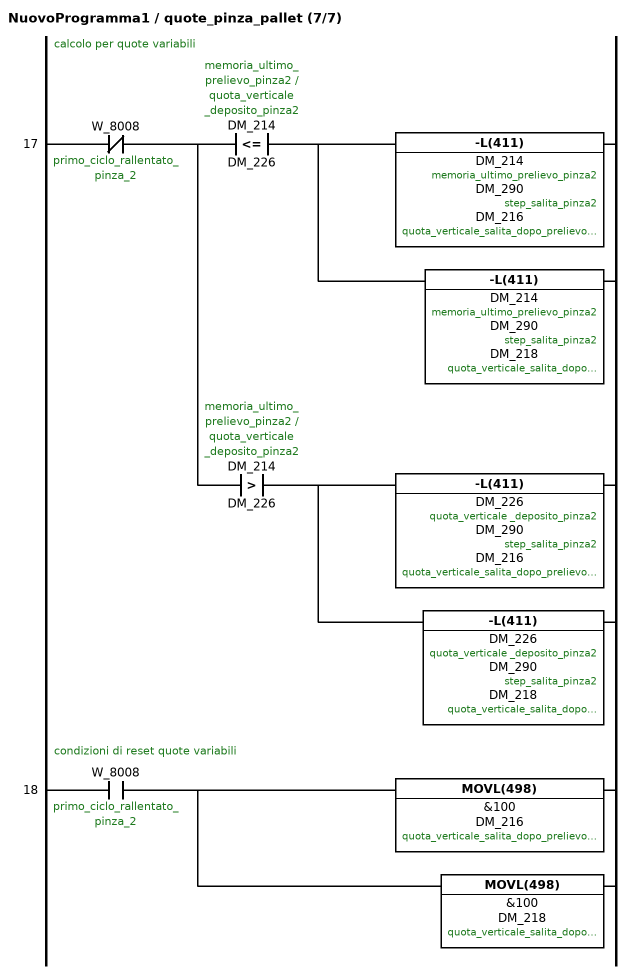
; [picture p96: NuovoProgramma1 / quote_pinza_pallet, rungs 17-18]
; rung 17: calcolo per quote variabili
LDNOT W_8008  ; primo_ciclo_rallentato_pinza_2
OUT TR0
AND<=SL(318) DM_214 DM_226  ; memoria_ultimo_prelievo_pinza2, quota_verticale _deposito_pinza2
-L(411) DM_214 DM_290 DM_216  ; memoria_ultimo_prelievo_pinza2, step_salita_pinza2, quota_verticale_salita_dopo_prelievo_pinza2
-L(411) DM_214 DM_290 DM_218  ; memoria_ultimo_prelievo_pinza2, step_salita_pinza2, quota_verticale_salita_dopo_deposito_pinza2
LD TR0
AND>SL(323) DM_214 DM_226  ; memoria_ultimo_prelievo_pinza2, quota_verticale _deposito_pinza2
-L(411) DM_226 DM_290 DM_216  ; quota_verticale _deposito_pinza2, step_salita_pinza2, quota_verticale_salita_dopo_prelievo_pinza2
-L(411) DM_226 DM_290 DM_218  ; quota_verticale _deposito_pinza2, step_salita_pinza2, quota_verticale_salita_dopo_deposito_pinza2
; rung 18: condizioni di reset quote variabili
LD W_8008  ; primo_ciclo_rallentato_pinza_2
MOVL(498) &100 DM_216  ; quota_verticale_salita_dopo_prelievo_pinza2
MOVL(498) &100 DM_218  ; quota_verticale_salita_dopo_deposito_pinza2

### Section cambi_pallet

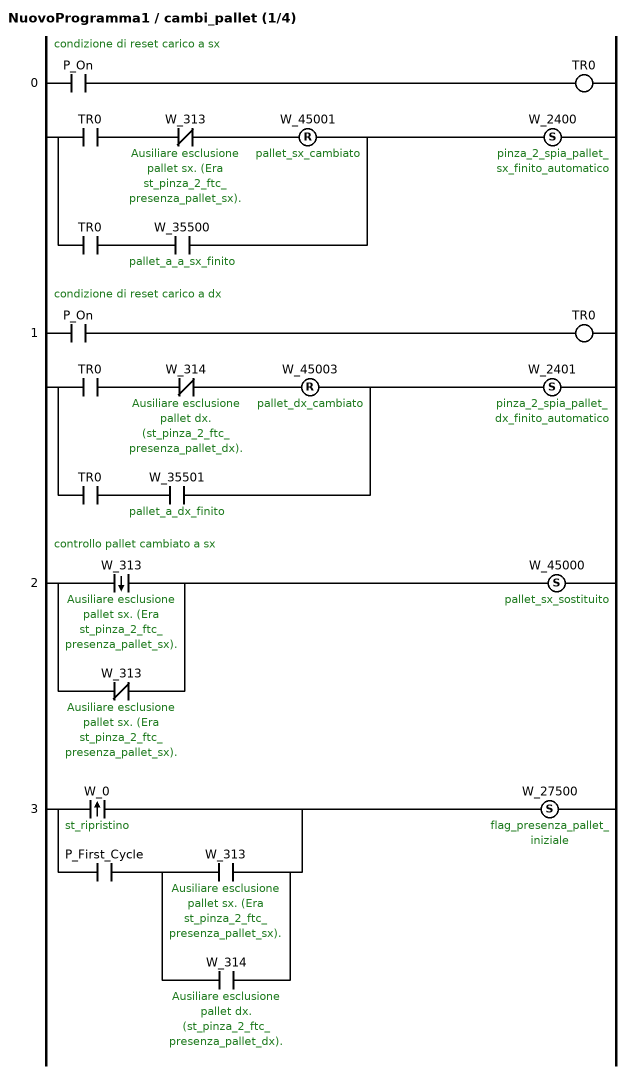
; rung 0: condizione di reset carico a sx
LD P_On
OUT TR0
ANDNOT W_313  ; Ausiliare esclusione pallet sx. (Era st_pinza_2_ftc_presenza_pallet_sx).
RSET W_45001  ; pallet_sx_cambiato
LD TR0
AND W_35500  ; pallet_a_a_sx_finito
ORLD
SET W_2400  ; pinza_2_spia_pallet_sx_finito_automatico
; rung 1: condizione di reset carico a dx
LD P_On
OUT TR0
ANDNOT W_314  ; Ausiliare esclusione pallet dx. (st_pinza_2_ftc_presenza_pallet_dx).
RSET W_45003  ; pallet_dx_cambiato
LD TR0
AND W_35501  ; pallet_a_dx_finito
ORLD
SET W_2401  ; pinza_2_spia_pallet_dx_finito_automatico
; rung 2: controllo pallet cambiato a sx
%LD W_313  ; Ausiliare esclusione pallet sx. (Era st_pinza_2_ftc_presenza_pallet_sx).
ORNOT W_313  ; Ausiliare esclusione pallet sx. (Era st_pinza_2_ftc_presenza_pallet_sx).
SET W_45000  ; pallet_sx_sostituito
; rung 3
@LD W_0  ; st_ripristino
LD P_First_Cycle
LD W_313  ; Ausiliare esclusione pallet sx. (Era st_pinza_2_ftc_presenza_pallet_sx).
OR W_314  ; Ausiliare esclusione pallet dx. (st_pinza_2_ftc_presenza_pallet_dx).
ANDLD
ORLD
SET W_27500  ; flag_presenza_pallet_iniziale

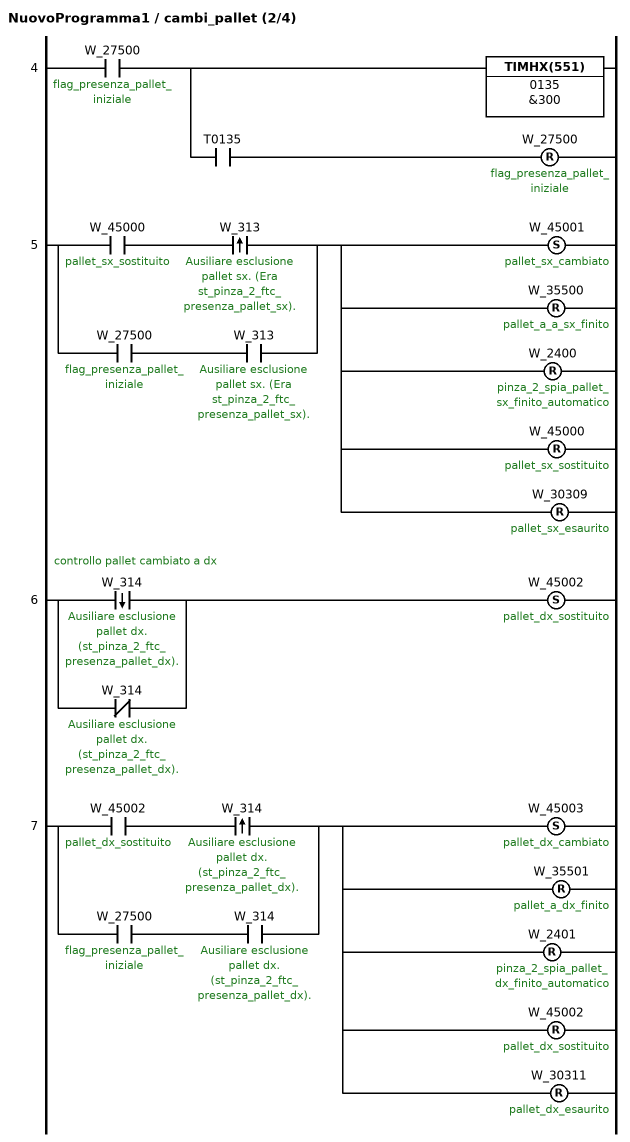
; rung 4
LD W_27500  ; flag_presenza_pallet_iniziale
TIMHX(551) 0135 &300
AND T0135
RSET W_27500  ; flag_presenza_pallet_iniziale
; rung 5
LD W_45000  ; pallet_sx_sostituito
@AND W_313  ; Ausiliare esclusione pallet sx. (Era st_pinza_2_ftc_presenza_pallet_sx).
LD W_27500  ; flag_presenza_pallet_iniziale
AND W_313  ; Ausiliare esclusione pallet sx. (Era st_pinza_2_ftc_presenza_pallet_sx).
ORLD
SET W_45001  ; pallet_sx_cambiato
RSET W_35500  ; pallet_a_a_sx_finito
RSET W_2400  ; pinza_2_spia_pallet_sx_finito_automatico
RSET W_45000  ; pallet_sx_sostituito
RSET W_30309  ; pallet_sx_esaurito
; rung 6: controllo pallet cambiato a dx
%LD W_314  ; Ausiliare esclusione pallet dx. (st_pinza_2_ftc_presenza_pallet_dx).
ORNOT W_314  ; Ausiliare esclusione pallet dx. (st_pinza_2_ftc_presenza_pallet_dx).
SET W_45002  ; pallet_dx_sostituito
; rung 7
LD W_45002  ; pallet_dx_sostituito
@AND W_314  ; Ausiliare esclusione pallet dx. (st_pinza_2_ftc_presenza_pallet_dx).
LD W_27500  ; flag_presenza_pallet_iniziale
AND W_314  ; Ausiliare esclusione pallet dx. (st_pinza_2_ftc_presenza_pallet_dx).
ORLD
SET W_45003  ; pallet_dx_cambiato
RSET W_35501  ; pallet_a_dx_finito
RSET W_2401  ; pinza_2_spia_pallet_dx_finito_automatico
RSET W_45002  ; pallet_dx_sostituito
RSET W_30311  ; pallet_dx_esaurito

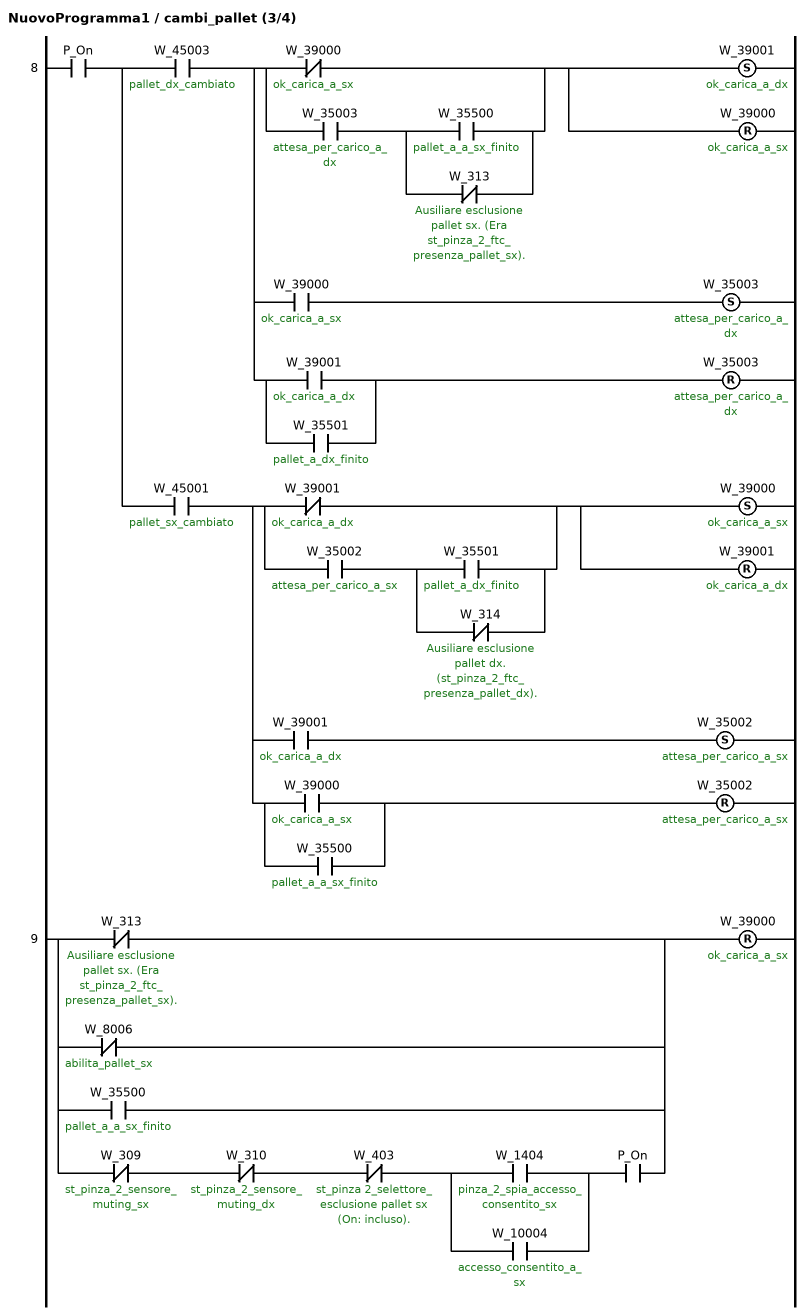
; rung 8
LD P_On
OUT TR0
AND W_45003  ; pallet_dx_cambiato
OUT TR1
LDNOT W_39000  ; ok_carica_a_sx
LD W_35003  ; attesa_per_carico_a_dx
LD W_35500  ; pallet_a_a_sx_finito
ORNOT W_313  ; Ausiliare esclusione pallet sx. (Era st_pinza_2_ftc_presenza_pallet_sx).
ANDLD
ORLD
ANDLD
SET W_39001  ; ok_carica_a_dx
RSET W_39000  ; ok_carica_a_sx
LD TR1
AND W_39000  ; ok_carica_a_sx
SET W_35003  ; attesa_per_carico_a_dx
LD TR1
LD W_39001  ; ok_carica_a_dx
OR W_35501  ; pallet_a_dx_finito
ANDLD
RSET W_35003  ; attesa_per_carico_a_dx
LD TR0
AND W_45001  ; pallet_sx_cambiato
OUT TR0
LDNOT W_39001  ; ok_carica_a_dx
LD W_35002  ; attesa_per_carico_a_sx
LD W_35501  ; pallet_a_dx_finito
ORNOT W_314  ; Ausiliare esclusione pallet dx. (st_pinza_2_ftc_presenza_pallet_dx).
ANDLD
ORLD
ANDLD
SET W_39000  ; ok_carica_a_sx
RSET W_39001  ; ok_carica_a_dx
LD TR0
AND W_39001  ; ok_carica_a_dx
SET W_35002  ; attesa_per_carico_a_sx
LD TR0
LD W_39000  ; ok_carica_a_sx
OR W_35500  ; pallet_a_a_sx_finito
ANDLD
RSET W_35002  ; attesa_per_carico_a_sx
; rung 9
LDNOT W_313  ; Ausiliare esclusione pallet sx. (Era st_pinza_2_ftc_presenza_pallet_sx).
ORNOT W_8006  ; abilita_pallet_sx
OR W_35500  ; pallet_a_a_sx_finito
LDNOT W_309  ; st_pinza_2_sensore_muting_sx
ANDNOT W_310  ; st_pinza_2_sensore_muting_dx
ANDNOT W_403  ; st_pinza 2_selettore_esclusione pallet sx (On: incluso).
LD W_1404  ; pinza_2_spia_accesso_consentito_sx
OR W_10004  ; accesso_consentito_a_sx
ANDLD
AND P_On
ORLD
RSET W_39000  ; ok_carica_a_sx

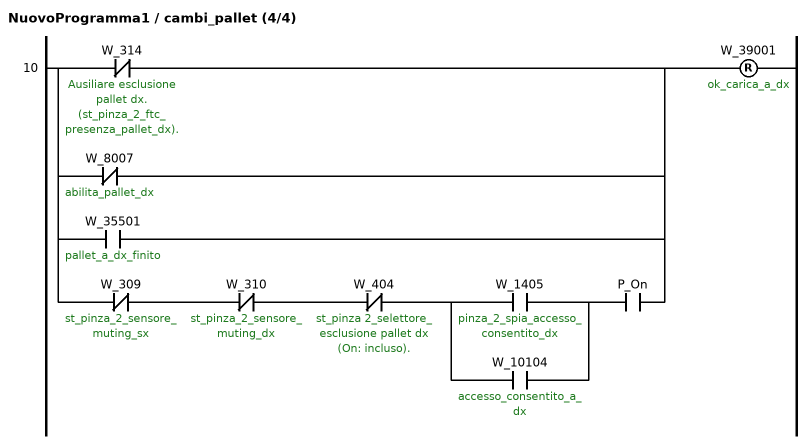
; rung 10
LDNOT W_314  ; Ausiliare esclusione pallet dx. (st_pinza_2_ftc_presenza_pallet_dx).
ORNOT W_8007  ; abilita_pallet_dx
OR W_35501  ; pallet_a_dx_finito
LDNOT W_309  ; st_pinza_2_sensore_muting_sx
ANDNOT W_310  ; st_pinza_2_sensore_muting_dx
ANDNOT W_404  ; st_pinza 2_selettore_esclusione pallet dx (On: incluso).
LD W_1405  ; pinza_2_spia_accesso_consentito_dx
OR W_10104  ; accesso_consentito_a_dx
ANDLD
AND P_On
ORLD
RSET W_39001  ; ok_carica_a_dx

### Section accessi

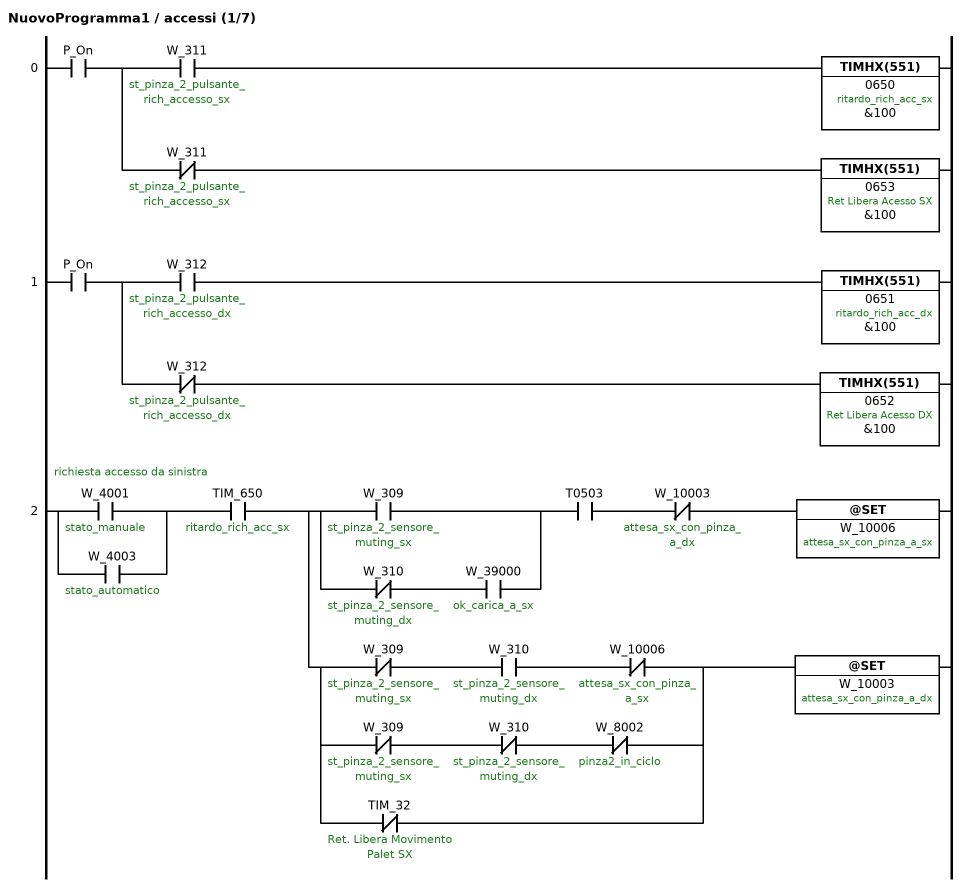
; rung 0
LD P_On
OUT TR0
AND W_311  ; st_pinza_2_pulsante_rich_accesso_sx
TIMHX(551) 0650 &100  ; ritardo_rich_acc_sx
LD TR0
ANDNOT W_311  ; st_pinza_2_pulsante_rich_accesso_sx
TIMHX(551) 0653 &100  ; Ret Libera Acesso SX
; rung 1
LD P_On
OUT TR0
AND W_312  ; st_pinza_2_pulsante_rich_accesso_dx
TIMHX(551) 0651 &100  ; ritardo_rich_acc_dx
LD TR0
ANDNOT W_312  ; st_pinza_2_pulsante_rich_accesso_dx
TIMHX(551) 0652 &100  ; Ret Libera Acesso DX
; rung 2: richiesta accesso da sinistra
LD W_4001  ; stato_manuale
OR W_4003  ; stato_automatico
AND TIM_650  ; ritardo_rich_acc_sx
OUT TR0
LD W_309  ; st_pinza_2_sensore_muting_sx
LDNOT W_310  ; st_pinza_2_sensore_muting_dx
AND W_39000  ; ok_carica_a_sx
ORLD
ANDLD
AND T0503
ANDNOT W_10003  ; attesa_sx_con_pinza_a_dx
@SET W_10006  ; attesa_sx_con_pinza_a_sx
LD TR0
LDNOT W_309  ; st_pinza_2_sensore_muting_sx
AND W_310  ; st_pinza_2_sensore_muting_dx
ANDNOT W_10006  ; attesa_sx_con_pinza_a_sx
LDNOT W_309  ; st_pinza_2_sensore_muting_sx
ANDNOT W_310  ; st_pinza_2_sensore_muting_dx
ANDNOT W_8002  ; pinza2_in_ciclo
ORLD
ORNOT TIM_32  ; Ret. Libera Movimento Palet SX
ANDLD
@SET W_10003  ; attesa_sx_con_pinza_a_dx

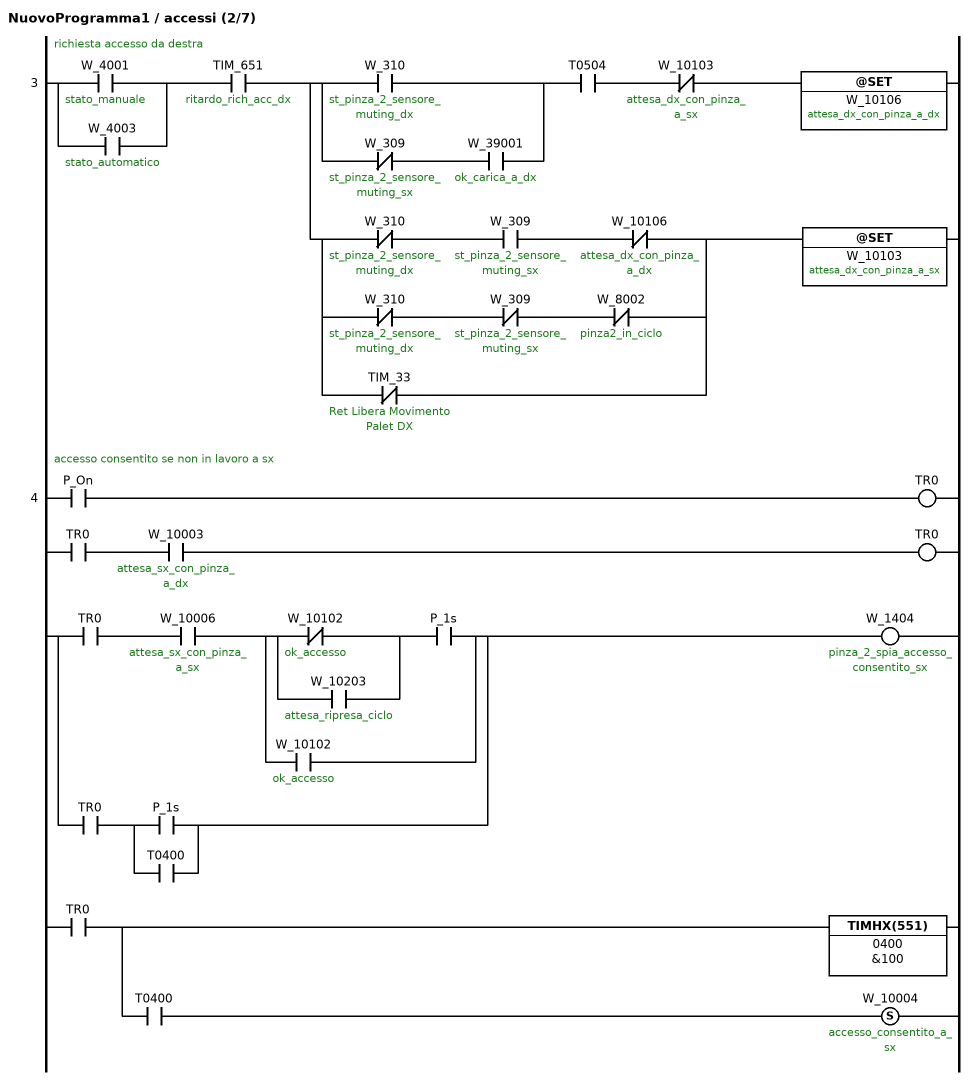
; rung 3: richiesta accesso da destra
LD W_4001  ; stato_manuale
OR W_4003  ; stato_automatico
AND TIM_651  ; ritardo_rich_acc_dx
OUT TR0
LD W_310  ; st_pinza_2_sensore_muting_dx
LDNOT W_309  ; st_pinza_2_sensore_muting_sx
AND W_39001  ; ok_carica_a_dx
ORLD
ANDLD
AND T0504
ANDNOT W_10103  ; attesa_dx_con_pinza_a_sx
@SET W_10106  ; attesa_dx_con_pinza_a_dx
LD TR0
LDNOT W_310  ; st_pinza_2_sensore_muting_dx
AND W_309  ; st_pinza_2_sensore_muting_sx
ANDNOT W_10106  ; attesa_dx_con_pinza_a_dx
LDNOT W_310  ; st_pinza_2_sensore_muting_dx
ANDNOT W_309  ; st_pinza_2_sensore_muting_sx
ANDNOT W_8002  ; pinza2_in_ciclo
ORLD
ORNOT TIM_33  ; Ret Libera Movimento Palet DX
ANDLD
@SET W_10103  ; attesa_dx_con_pinza_a_sx
; rung 4: accesso consentito se non in lavoro a sx
LD P_On
OUT TR0
AND W_10006  ; attesa_sx_con_pinza_a_sx
LDNOT W_10102  ; ok_accesso
OR W_10203  ; attesa_ripresa_ciclo
AND P_1s
OR W_10102  ; ok_accesso
ANDLD
LD TR0
AND W_10003  ; attesa_sx_con_pinza_a_dx
OUT TR0
LD P_1s
OR T0400
ANDLD
ORLD
OUT W_1404  ; pinza_2_spia_accesso_consentito_sx
LD TR0
TIMHX(551) 0400 &100
AND T0400
SET W_10004  ; accesso_consentito_a_sx

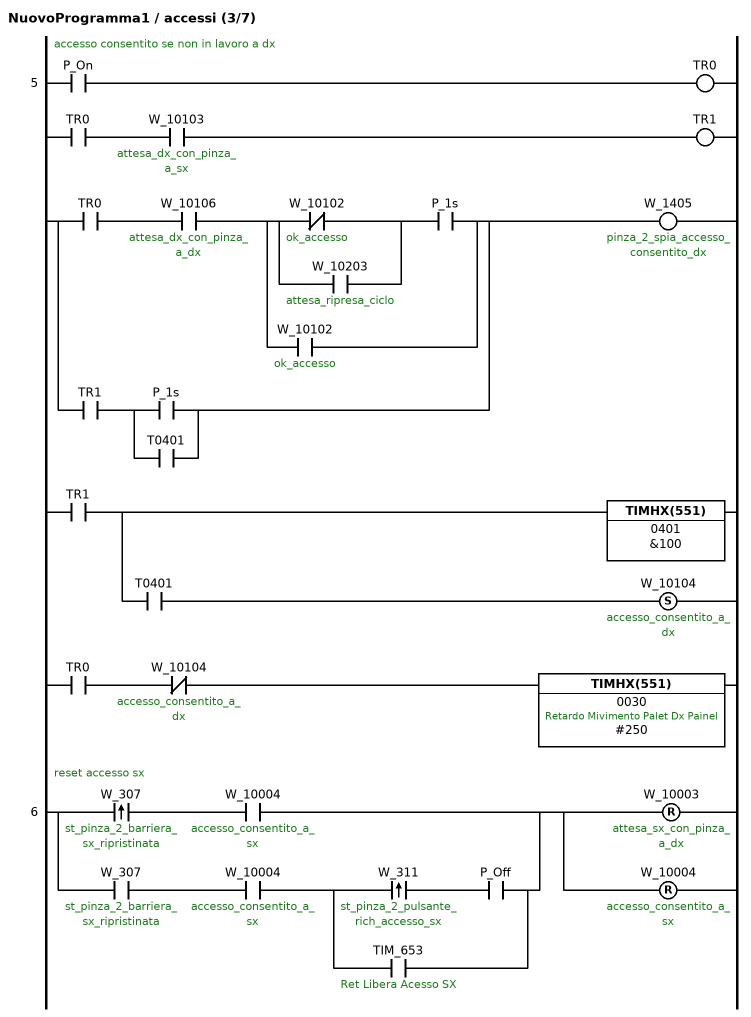
; rung 5: accesso consentito se non in lavoro a dx
LD P_On
OUT TR0
AND W_10106  ; attesa_dx_con_pinza_a_dx
LDNOT W_10102  ; ok_accesso
OR W_10203  ; attesa_ripresa_ciclo
AND P_1s
OR W_10102  ; ok_accesso
ANDLD
LD TR0
AND W_10103  ; attesa_dx_con_pinza_a_sx
OUT TR1
LD P_1s
OR T0401
ANDLD
ORLD
OUT W_1405  ; pinza_2_spia_accesso_consentito_dx
LD TR1
TIMHX(551) 0401 &100
AND T0401
SET W_10104  ; accesso_consentito_a_dx
LD TR0
ANDNOT W_10104  ; accesso_consentito_a_dx
TIMHX(551) 0030 #250  ; Retardo Mivimento Palet Dx Painel
; rung 6: reset accesso sx
@LD W_307  ; st_pinza_2_barriera_sx_ripristinata
AND W_10004  ; accesso_consentito_a_sx
LD W_307  ; st_pinza_2_barriera_sx_ripristinata
AND W_10004  ; accesso_consentito_a_sx
@LD W_311  ; st_pinza_2_pulsante_rich_accesso_sx
AND P_Off
OR TIM_653  ; Ret Libera Acesso SX
ANDLD
ORLD
RSET W_10003  ; attesa_sx_con_pinza_a_dx
RSET W_10004  ; accesso_consentito_a_sx

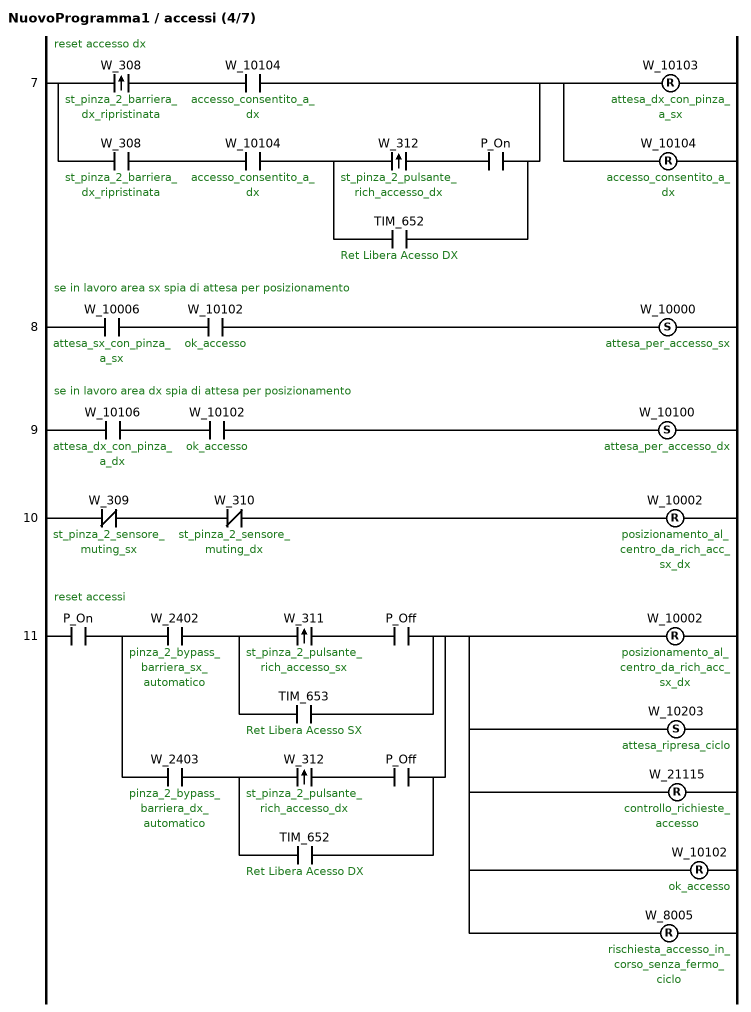
; rung 7: reset accesso dx
@LD W_308  ; st_pinza_2_barriera_dx_ripristinata
AND W_10104  ; accesso_consentito_a_dx
LD W_308  ; st_pinza_2_barriera_dx_ripristinata
AND W_10104  ; accesso_consentito_a_dx
@LD W_312  ; st_pinza_2_pulsante_rich_accesso_dx
AND P_On
OR TIM_652  ; Ret Libera Acesso DX
ANDLD
ORLD
RSET W_10103  ; attesa_dx_con_pinza_a_sx
RSET W_10104  ; accesso_consentito_a_dx
; rung 8: se in lavoro area sx spia di attesa per posizionamento
LD W_10006  ; attesa_sx_con_pinza_a_sx
AND W_10102  ; ok_accesso
SET W_10000  ; attesa_per_accesso_sx
; rung 9: se in lavoro area dx spia di attesa per posizionamento
LD W_10106  ; attesa_dx_con_pinza_a_dx
AND W_10102  ; ok_accesso
SET W_10100  ; attesa_per_accesso_dx
; rung 10
LDNOT W_309  ; st_pinza_2_sensore_muting_sx
ANDNOT W_310  ; st_pinza_2_sensore_muting_dx
RSET W_10002  ; posizionamento_al_centro_da_rich_acc_sx_dx
; rung 11: reset accessi
LD P_On
LD W_2402  ; pinza_2_bypass_barriera_sx_automatico
@LD W_311  ; st_pinza_2_pulsante_rich_accesso_sx
AND P_Off
OR TIM_653  ; Ret Libera Acesso SX
ANDLD
LD W_2403  ; pinza_2_bypass_barriera_dx_automatico
@LD W_312  ; st_pinza_2_pulsante_rich_accesso_dx
AND P_Off
OR TIM_652  ; Ret Libera Acesso DX
ANDLD
ORLD
ANDLD
RSET W_10002  ; posizionamento_al_centro_da_rich_acc_sx_dx
SET W_10203  ; attesa_ripresa_ciclo
RSET W_21115  ; controllo_richieste_accesso
RSET W_10102  ; ok_accesso
RSET W_8005  ; rischiesta_accesso_in_corso_senza_fermo_ciclo

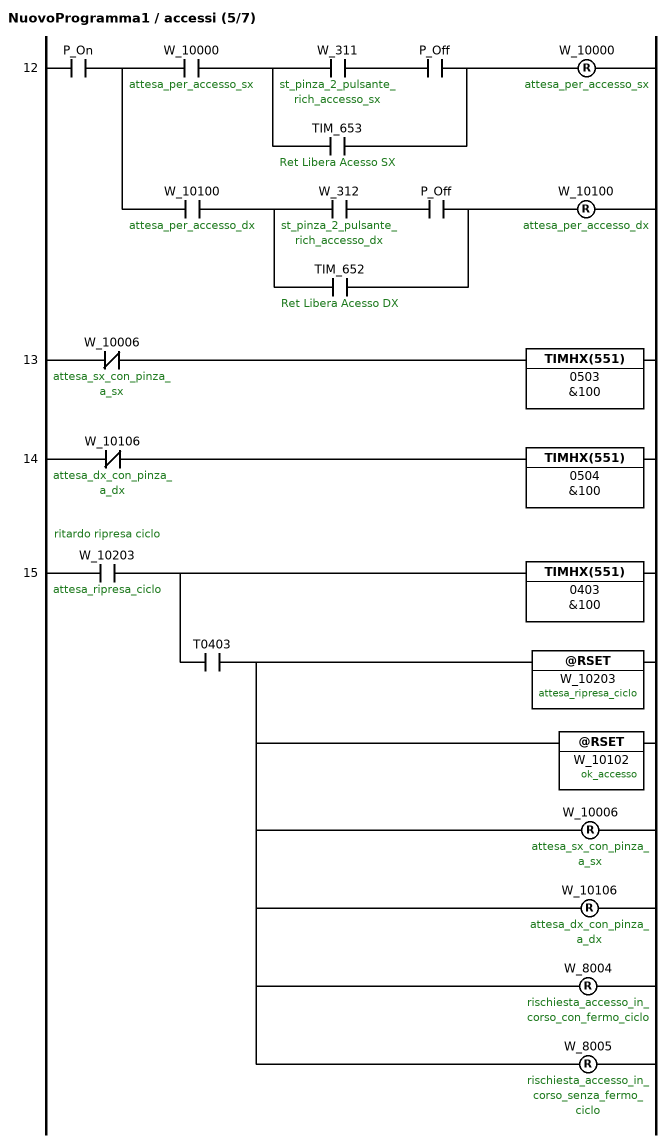
; rung 12
LD P_On
OUT TR0
AND W_10000  ; attesa_per_accesso_sx
LD W_311  ; st_pinza_2_pulsante_rich_accesso_sx
AND P_Off
OR TIM_653  ; Ret Libera Acesso SX
ANDLD
RSET W_10000  ; attesa_per_accesso_sx
LD TR0
AND W_10100  ; attesa_per_accesso_dx
LD W_312  ; st_pinza_2_pulsante_rich_accesso_dx
AND P_Off
OR TIM_652  ; Ret Libera Acesso DX
ANDLD
RSET W_10100  ; attesa_per_accesso_dx
; rung 13
LDNOT W_10006  ; attesa_sx_con_pinza_a_sx
TIMHX(551) 0503 &100
; rung 14
LDNOT W_10106  ; attesa_dx_con_pinza_a_dx
TIMHX(551) 0504 &100
; rung 15: ritardo ripresa ciclo
LD W_10203  ; attesa_ripresa_ciclo
TIMHX(551) 0403 &100
AND T0403
@RSET W_10203  ; attesa_ripresa_ciclo
@RSET W_10102  ; ok_accesso
RSET W_10006  ; attesa_sx_con_pinza_a_sx
RSET W_10106  ; attesa_dx_con_pinza_a_dx
RSET W_8004  ; rischiesta_accesso_in_corso_con_fermo_ciclo
RSET W_8005  ; rischiesta_accesso_in_corso_senza_fermo_ciclo

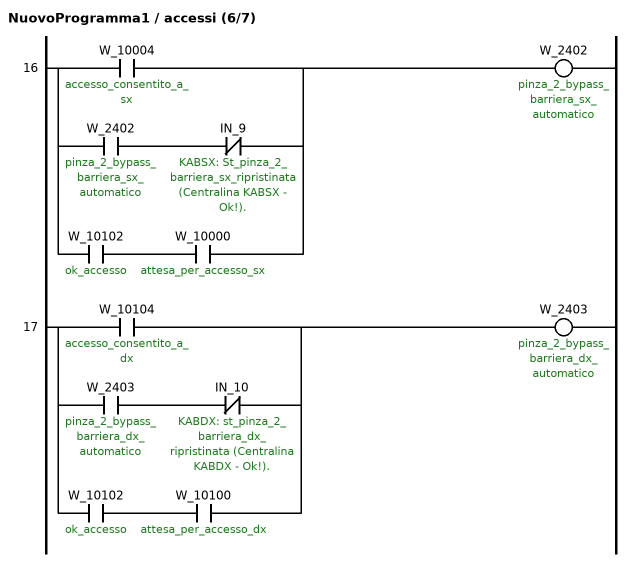
; rung 16
LD W_10004  ; accesso_consentito_a_sx
LD W_2402  ; pinza_2_bypass_barriera_sx_automatico
ANDNOT IN_9  ; KABSX: St_pinza_2_barriera_sx_ripristinata (Centralina KABSX - Ok!).
ORLD
LD W_10102  ; ok_accesso
AND W_10000  ; attesa_per_accesso_sx
ORLD
OUT W_2402  ; pinza_2_bypass_barriera_sx_automatico
; rung 17
LD W_10104  ; accesso_consentito_a_dx
LD W_2403  ; pinza_2_bypass_barriera_dx_automatico
ANDNOT IN_10  ; KABDX: st_pinza_2_barriera_dx_ripristinata (Centralina KABDX - Ok!).
ORLD
LD W_10102  ; ok_accesso
AND W_10100  ; attesa_per_accesso_dx
ORLD
OUT W_2403  ; pinza_2_bypass_barriera_dx_automatico

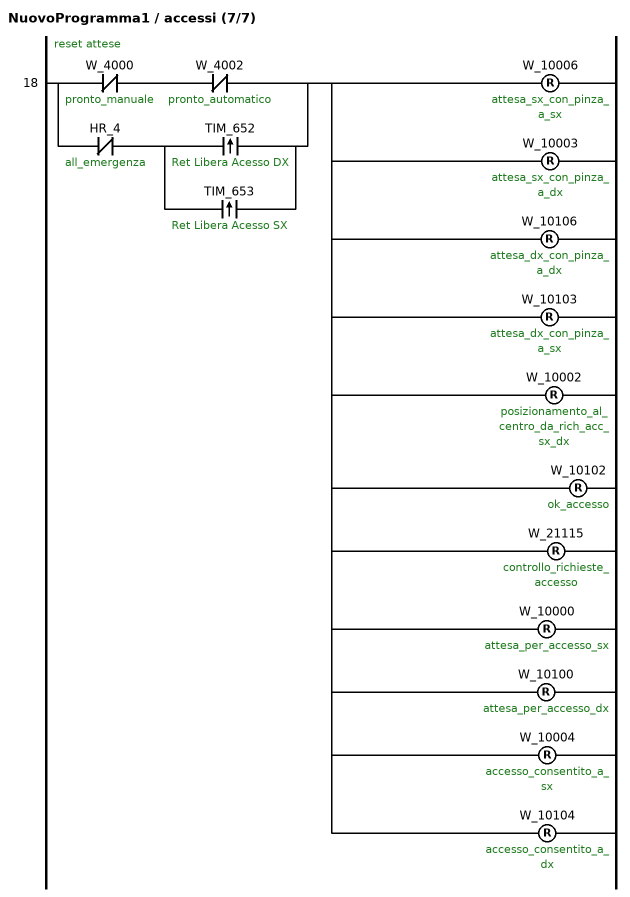
; rung 18: reset attese
LDNOT W_4000  ; pronto_manuale
ANDNOT W_4002  ; pronto_automatico
LDNOT HR_4  ; all_emergenza
@LD TIM_652  ; Ret Libera Acesso DX
@OR TIM_653  ; Ret Libera Acesso SX
ANDLD
ORLD
RSET W_10006  ; attesa_sx_con_pinza_a_sx
RSET W_10003  ; attesa_sx_con_pinza_a_dx
RSET W_10106  ; attesa_dx_con_pinza_a_dx
RSET W_10103  ; attesa_dx_con_pinza_a_sx
RSET W_10002  ; posizionamento_al_centro_da_rich_acc_sx_dx
RSET W_10102  ; ok_accesso
RSET W_21115  ; controllo_richieste_accesso
RSET W_10000  ; attesa_per_accesso_sx
RSET W_10100  ; attesa_per_accesso_dx
RSET W_10004  ; accesso_consentito_a_sx
RSET W_10104  ; accesso_consentito_a_dx

### Section inverter

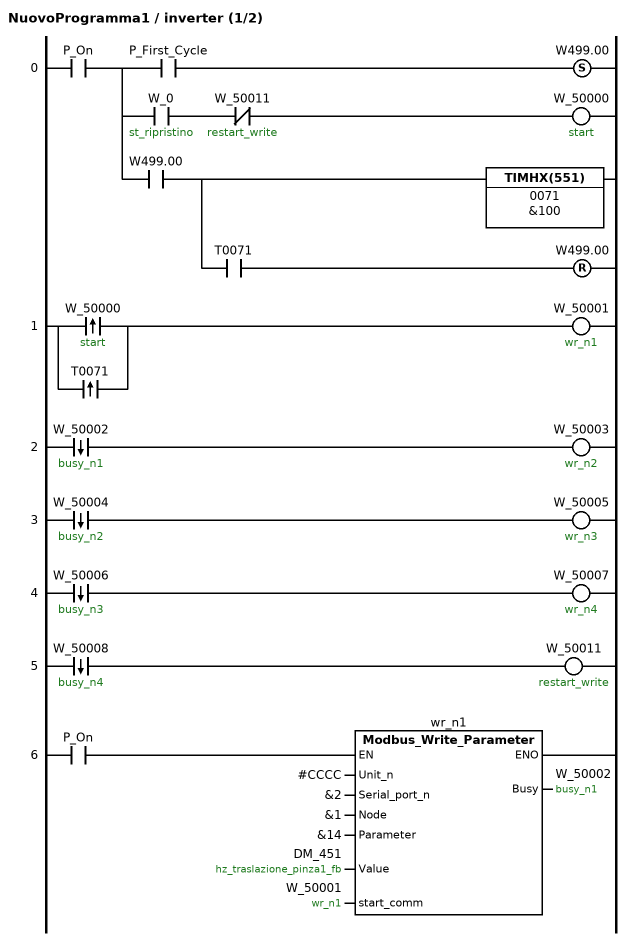
; rung 0
LD P_On
OUT TR0
AND P_First_Cycle
SET W499.00
LD TR0
AND W_0  ; st_ripristino
ANDNOT W_50011  ; restart_write
OUT W_50000  ; start
LD TR0
AND W499.00
TIMHX(551) 0071 &100
AND T0071
RSET W499.00
; rung 1
@LD W_50000  ; start
@OR T0071
OUT W_50001  ; wr_n1
; rung 2
%LD W_50002  ; busy_n1
OUT W_50003  ; wr_n2
; rung 3
%LD W_50004  ; busy_n2
OUT W_50005  ; wr_n3
; rung 4
%LD W_50006  ; busy_n3
OUT W_50007  ; wr_n4
; rung 5
%LD W_50008  ; busy_n4
OUT W_50011  ; restart_write
; rung 6
LD P_On
CALL wr_n1 : Modbus_Write_Parameter (Unit_n := #CCCC, Serial_port_n := &2, Node := &1, Parameter := &14, Value := DM_451, start_comm := W_50001, Busy => W_50002)  ; hz_traslazione_pinza1_fb, wr_n1, busy_n1

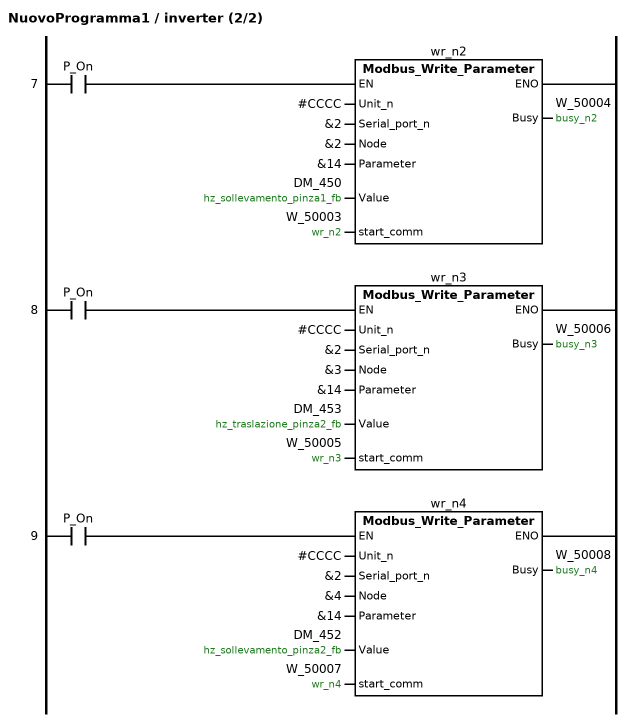
; rung 7
LD P_On
CALL wr_n2 : Modbus_Write_Parameter (Unit_n := #CCCC, Serial_port_n := &2, Node := &2, Parameter := &14, Value := DM_450, start_comm := W_50003, Busy => W_50004)  ; hz_sollevamento_pinza1_fb, wr_n2, busy_n2
; rung 8
LD P_On
CALL wr_n3 : Modbus_Write_Parameter (Unit_n := #CCCC, Serial_port_n := &2, Node := &3, Parameter := &14, Value := DM_453, start_comm := W_50005, Busy => W_50006)  ; hz_traslazione_pinza2_fb, wr_n3, busy_n3
; rung 9
LD P_On
CALL wr_n4 : Modbus_Write_Parameter (Unit_n := #CCCC, Serial_port_n := &2, Node := &4, Parameter := &14, Value := DM_452, start_comm := W_50007, Busy => W_50008)  ; hz_sollevamento_pinza2_fb, wr_n4, busy_n4

### Section allarmi

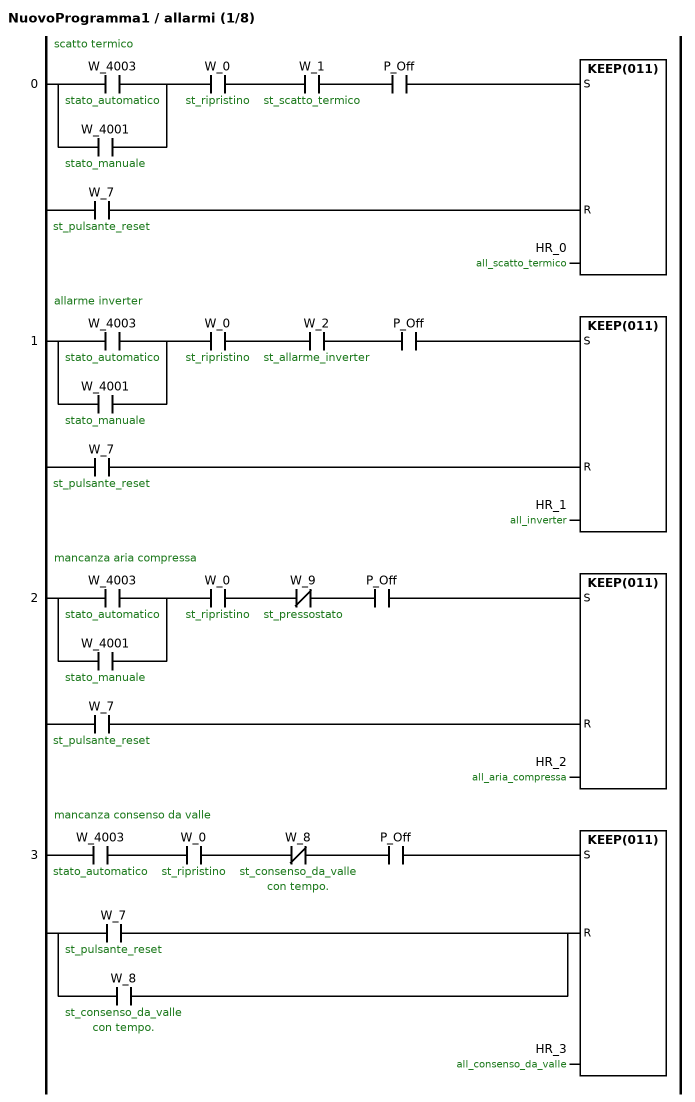
; rung 0: scatto termico
LD W_4003  ; stato_automatico
OR W_4001  ; stato_manuale
AND W_0  ; st_ripristino
AND W_1  ; st_scatto_termico
AND P_Off
LD W_7  ; st_pulsante_reset
KEEP(011) HR_0  ; all_scatto_termico
; rung 1: allarme inverter
LD W_4003  ; stato_automatico
OR W_4001  ; stato_manuale
AND W_0  ; st_ripristino
AND W_2  ; st_allarme_inverter
AND P_Off
LD W_7  ; st_pulsante_reset
KEEP(011) HR_1  ; all_inverter
; rung 2: mancanza aria compressa
LD W_4003  ; stato_automatico
OR W_4001  ; stato_manuale
AND W_0  ; st_ripristino
ANDNOT W_9  ; st_pressostato
AND P_Off
LD W_7  ; st_pulsante_reset
KEEP(011) HR_2  ; all_aria_compressa
; rung 3: mancanza consenso da valle
LD W_4003  ; stato_automatico
AND W_0  ; st_ripristino
ANDNOT W_8  ; st_consenso_da_valle con tempo.
AND P_Off
LD W_7  ; st_pulsante_reset
OR W_8  ; st_consenso_da_valle con tempo.
KEEP(011) HR_3  ; all_consenso_da_valle

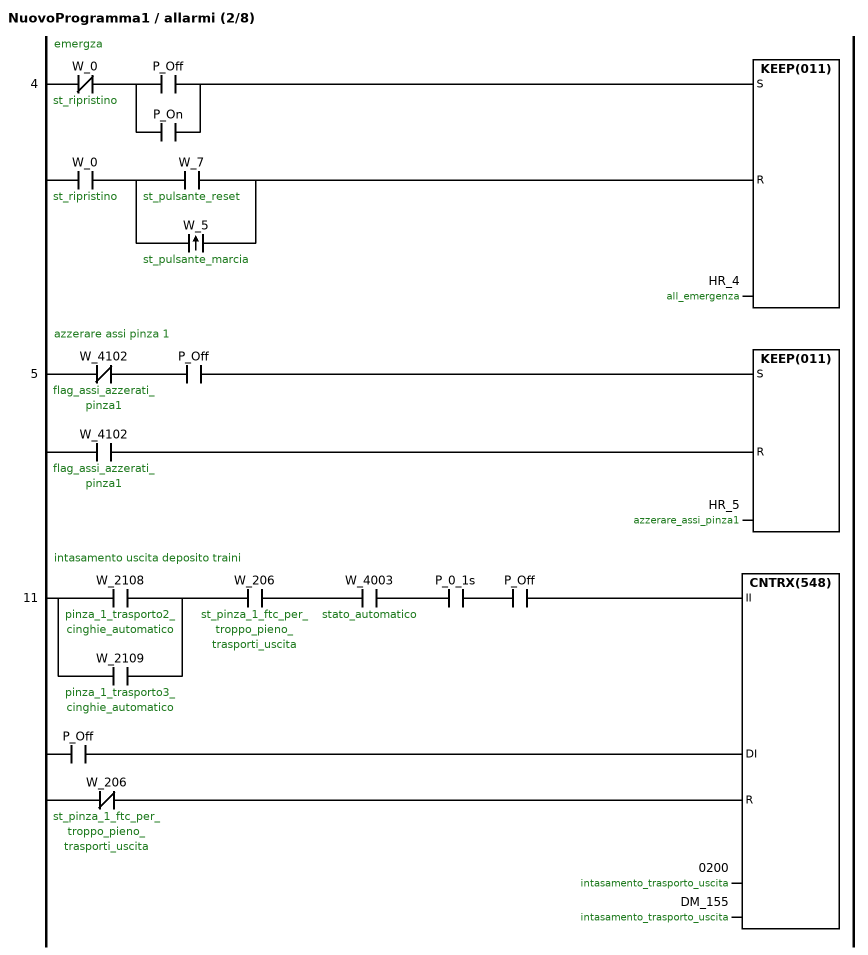
; rung 4: emergza
LDNOT W_0  ; st_ripristino
LD P_Off
OR P_On
ANDLD
LD W_0  ; st_ripristino
LD W_7  ; st_pulsante_reset
@OR W_5  ; st_pulsante_marcia
ANDLD
KEEP(011) HR_4  ; all_emergenza
; rung 5: azzerare assi pinza 1
LDNOT W_4102  ; flag_assi_azzerati_pinza1
AND P_Off
LD W_4102  ; flag_assi_azzerati_pinza1
KEEP(011) HR_5  ; azzerare_assi_pinza1
; rung 6: sensori tasteggio pinza 1
; rung 7: finecorsa basso pinza 1
; rung 8: encoder traslazione pinza 1
; rung 9: encoder sollevamento pinza 1
; rung 10: intasamento deposito traini
; rung 11: intasamento uscita deposito traini
LD W_2108  ; pinza_1_trasporto2_cinghie_automatico
OR W_2109  ; pinza_1_trasporto3_cinghie_automatico
AND W_206  ; st_pinza_1_ftc_per_troppo_pieno_trasporti_uscita
AND W_4003  ; stato_automatico
AND P_0_1s
AND P_Off
LD P_Off
LDNOT W_206  ; st_pinza_1_ftc_per_troppo_pieno_trasporti_uscita
CNTRX(548) 0200 DM_155  ; intasamento_trasporto_uscita

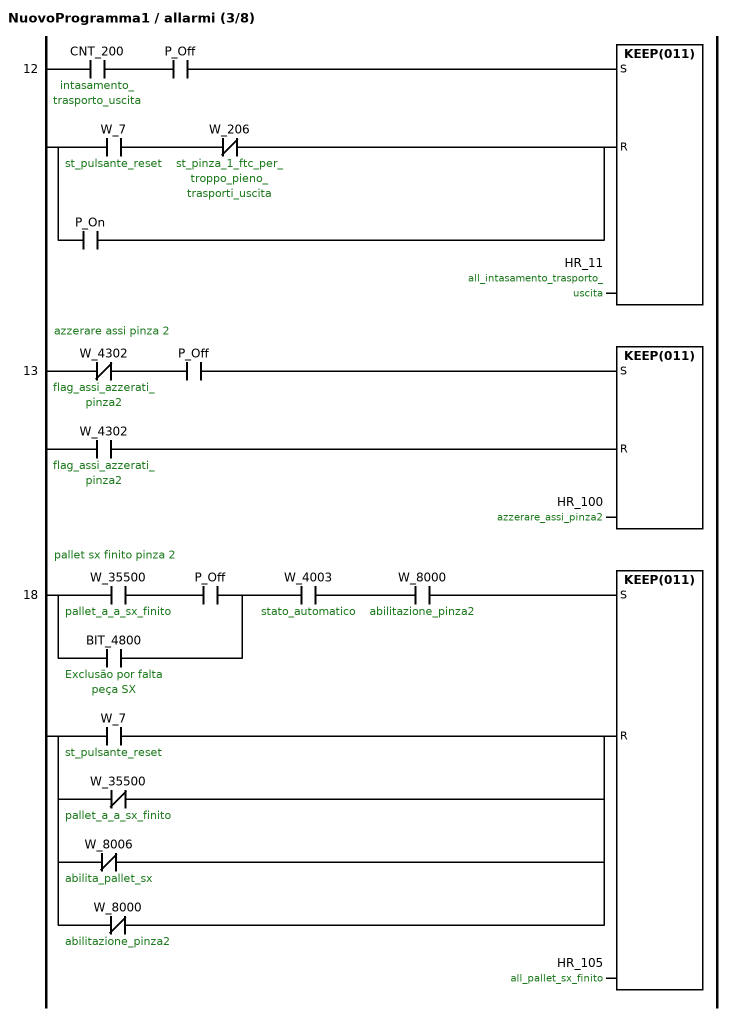
; rung 12
LD CNT_200  ; intasamento_trasporto_uscita
AND P_Off
LD W_7  ; st_pulsante_reset
ANDNOT W_206  ; st_pinza_1_ftc_per_troppo_pieno_trasporti_uscita
OR P_On
KEEP(011) HR_11  ; all_intasamento_trasporto_uscita
; rung 13: azzerare assi pinza 2
LDNOT W_4302  ; flag_assi_azzerati_pinza2
AND P_Off
LD W_4302  ; flag_assi_azzerati_pinza2
KEEP(011) HR_100  ; azzerare_assi_pinza2
; rung 14: sensori tasteggio pinza 2
; rung 15: finecorsa basso pinza 2
; rung 16: encoder traslazione pinza 2
; rung 17: encoder sollevamento pinza 2
; rung 18: pallet sx finito pinza 2
LD W_35500  ; pallet_a_a_sx_finito
AND P_Off
OR BIT_4800  ; Exclusão por falta peça SX
AND W_4003  ; stato_automatico
AND W_8000  ; abilitazione_pinza2
LD W_7  ; st_pulsante_reset
ORNOT W_35500  ; pallet_a_a_sx_finito
ORNOT W_8006  ; abilita_pallet_sx
ORNOT W_8000  ; abilitazione_pinza2
KEEP(011) HR_105  ; all_pallet_sx_finito

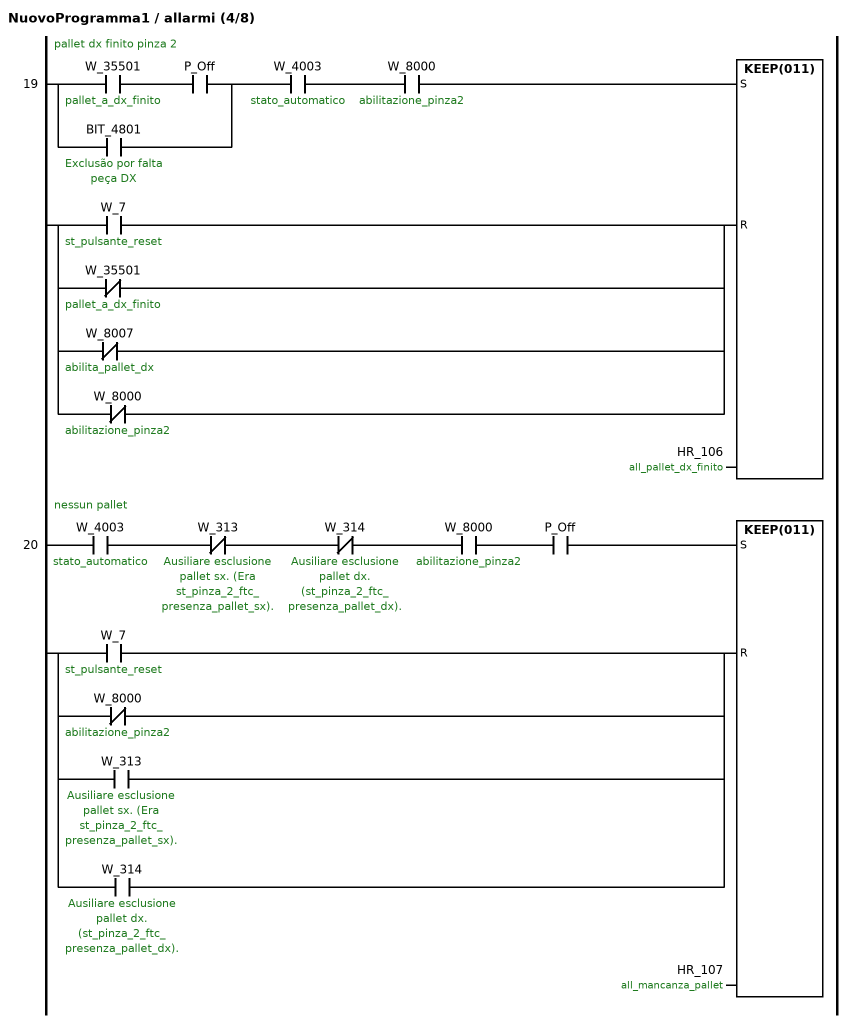
; rung 19: pallet dx finito pinza 2
LD W_35501  ; pallet_a_dx_finito
AND P_Off
OR BIT_4801  ; Exclusão por falta peça DX
AND W_4003  ; stato_automatico
AND W_8000  ; abilitazione_pinza2
LD W_7  ; st_pulsante_reset
ORNOT W_35501  ; pallet_a_dx_finito
ORNOT W_8007  ; abilita_pallet_dx
ORNOT W_8000  ; abilitazione_pinza2
KEEP(011) HR_106  ; all_pallet_dx_finito
; rung 20: nessun pallet
LD W_4003  ; stato_automatico
ANDNOT W_313  ; Ausiliare esclusione pallet sx. (Era st_pinza_2_ftc_presenza_pallet_sx).
ANDNOT W_314  ; Ausiliare esclusione pallet dx. (st_pinza_2_ftc_presenza_pallet_dx).
AND W_8000  ; abilitazione_pinza2
AND P_Off
LD W_7  ; st_pulsante_reset
ORNOT W_8000  ; abilitazione_pinza2
OR W_313  ; Ausiliare esclusione pallet sx. (Era st_pinza_2_ftc_presenza_pallet_sx).
OR W_314  ; Ausiliare esclusione pallet dx. (st_pinza_2_ftc_presenza_pallet_dx).
KEEP(011) HR_107  ; all_mancanza_pallet

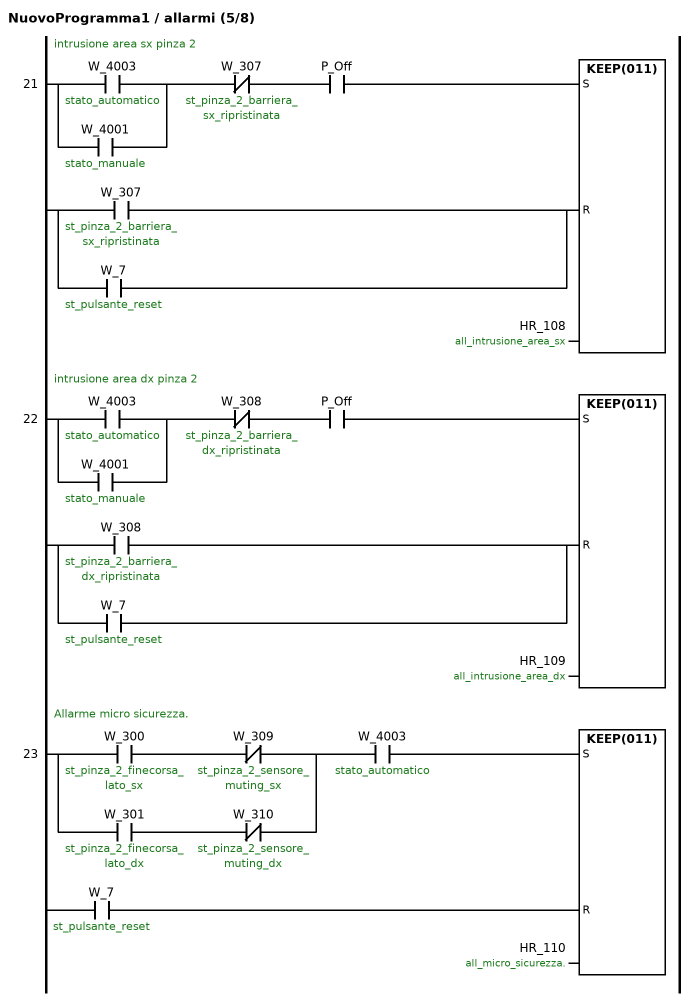
; rung 21: intrusione area sx pinza 2
LD W_4003  ; stato_automatico
OR W_4001  ; stato_manuale
ANDNOT W_307  ; st_pinza_2_barriera_sx_ripristinata
AND P_Off
LD W_307  ; st_pinza_2_barriera_sx_ripristinata
OR W_7  ; st_pulsante_reset
KEEP(011) HR_108  ; all_intrusione_area_sx
; rung 22: intrusione area dx pinza 2
LD W_4003  ; stato_automatico
OR W_4001  ; stato_manuale
ANDNOT W_308  ; st_pinza_2_barriera_dx_ripristinata
AND P_Off
LD W_308  ; st_pinza_2_barriera_dx_ripristinata
OR W_7  ; st_pulsante_reset
KEEP(011) HR_109  ; all_intrusione_area_dx
; rung 23: Allarme micro sicurezza.
LD W_300  ; st_pinza_2_finecorsa_lato_sx
ANDNOT W_309  ; st_pinza_2_sensore_muting_sx
LD W_301  ; st_pinza_2_finecorsa_lato_dx
ANDNOT W_310  ; st_pinza_2_sensore_muting_dx
ORLD
AND W_4003  ; stato_automatico
LD W_7  ; st_pulsante_reset
KEEP(011) HR_110  ; all_micro_sicurezza.

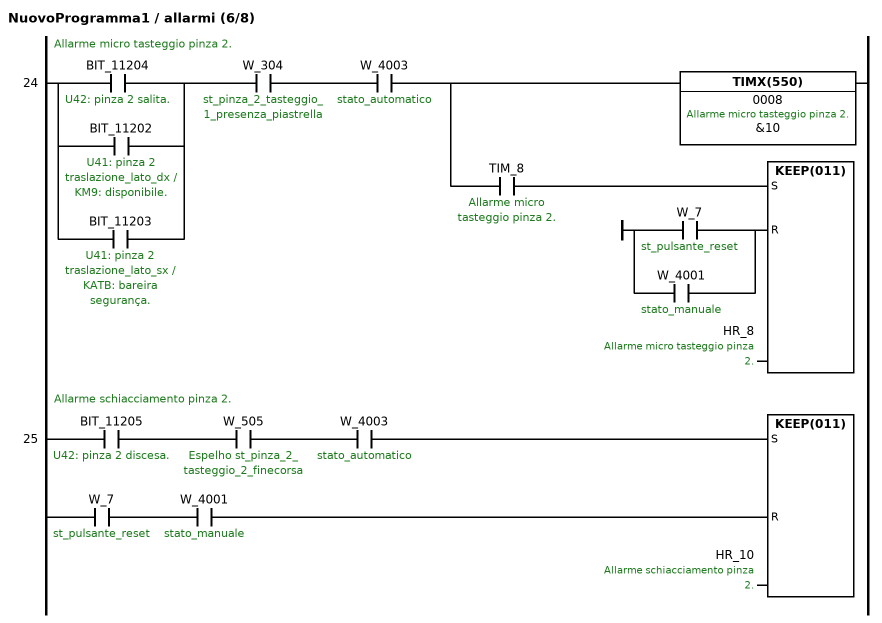
; rung 24: Allarme micro tasteggio pinza 2.
LD BIT_11204  ; U42: pinza 2 salita.
OR BIT_11202  ; U41: pinza 2 traslazione_lato_dx / KM9: disponibile.
OR BIT_11203  ; U41: pinza 2 traslazione_lato_sx / KATB: bareira segurança.
AND W_304  ; st_pinza_2_tasteggio_1_presenza_piastrella
AND W_4003  ; stato_automatico
TIMX(550) 0008 &10  ; Allarme micro tasteggio pinza 2.
AND TIM_8  ; Allarme micro tasteggio pinza 2.
LD W_7  ; st_pulsante_reset
OR W_4001  ; stato_manuale
KEEP(011) HR_8  ; Allarme micro tasteggio pinza 2.
; rung 25: Allarme schiacciamento pinza 2.
LD BIT_11205  ; U42: pinza 2 discesa.
AND W_505  ; Espelho st_pinza_2_tasteggio_2_finecorsa
AND W_4003  ; stato_automatico
LD W_7  ; st_pulsante_reset
AND W_4001  ; stato_manuale
KEEP(011) HR_10  ; Allarme schiacciamento pinza 2.

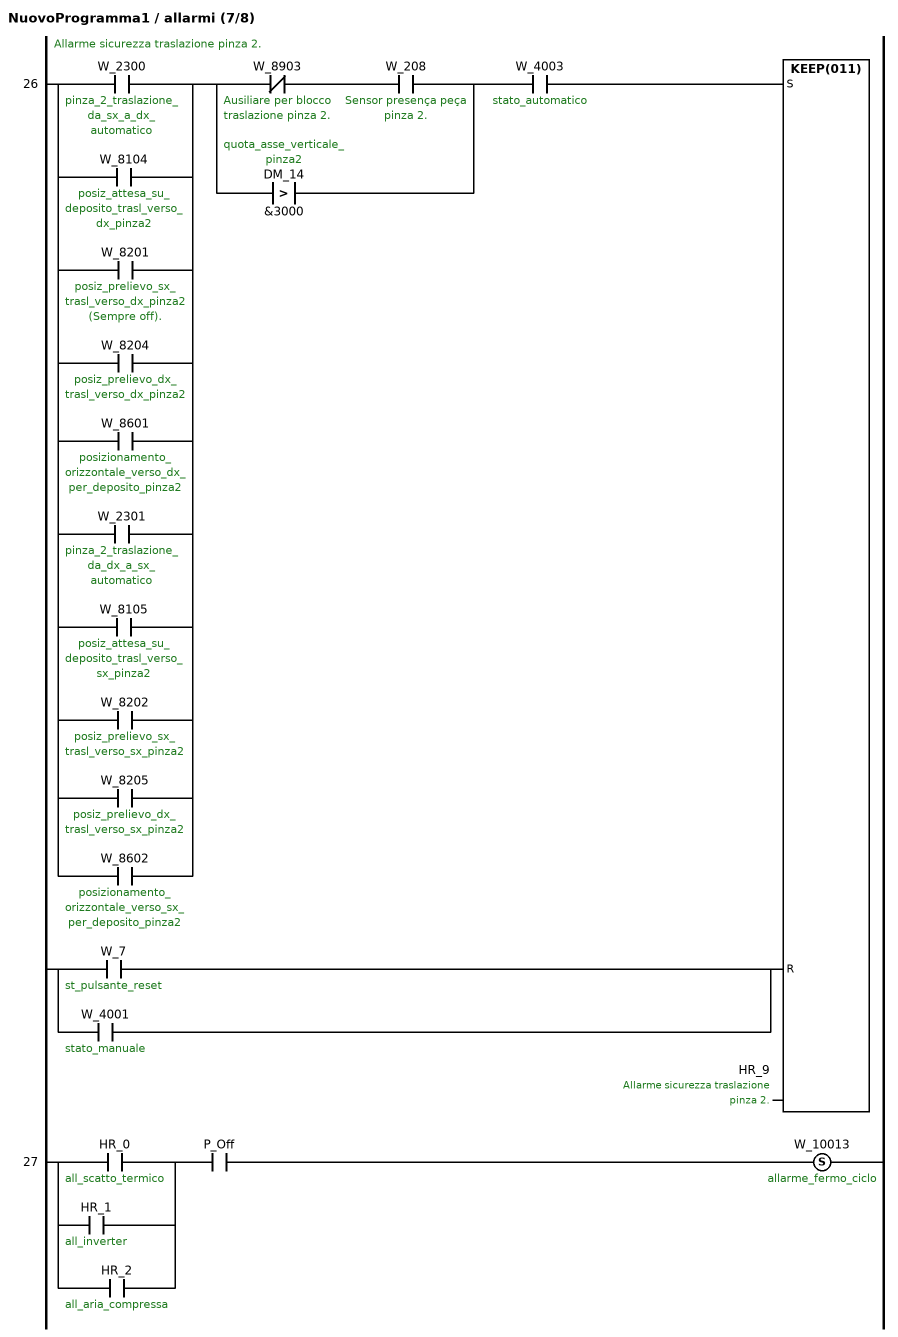
; rung 26: Allarme sicurezza traslazione pinza 2.
LD W_2300  ; pinza_2_traslazione_da_sx_a_dx_automatico
OR W_8104  ; posiz_attesa_su_deposito_trasl_verso_dx_pinza2
OR W_8201  ; posiz_prelievo_sx_trasl_verso_dx_pinza2 (Sempre off).
OR W_8204  ; posiz_prelievo_dx_trasl_verso_dx_pinza2
OR W_8601  ; posizionamento_orizzontale_verso_dx_per_deposito_pinza2
OR W_2301  ; pinza_2_traslazione_da_dx_a_sx_automatico
OR W_8105  ; posiz_attesa_su_deposito_trasl_verso_sx_pinza2
OR W_8202  ; posiz_prelievo_sx_trasl_verso_sx_pinza2
OR W_8205  ; posiz_prelievo_dx_trasl_verso_sx_pinza2
OR W_8602  ; posizionamento_orizzontale_verso_sx_per_deposito_pinza2
LDNOT W_8903  ; Ausiliare per blocco traslazione pinza 2.
AND W_208  ; Sensor presença peça pinza 2.
OR>S(322) DM_14 &3000  ; quota_asse_verticale_pinza2
ANDLD
AND W_4003  ; stato_automatico
LD W_7  ; st_pulsante_reset
OR W_4001  ; stato_manuale
KEEP(011) HR_9  ; Allarme sicurezza traslazione pinza 2.
; rung 27
LD HR_0  ; all_scatto_termico
OR HR_1  ; all_inverter
OR HR_2  ; all_aria_compressa
AND P_Off
SET W_10013  ; allarme_fermo_ciclo

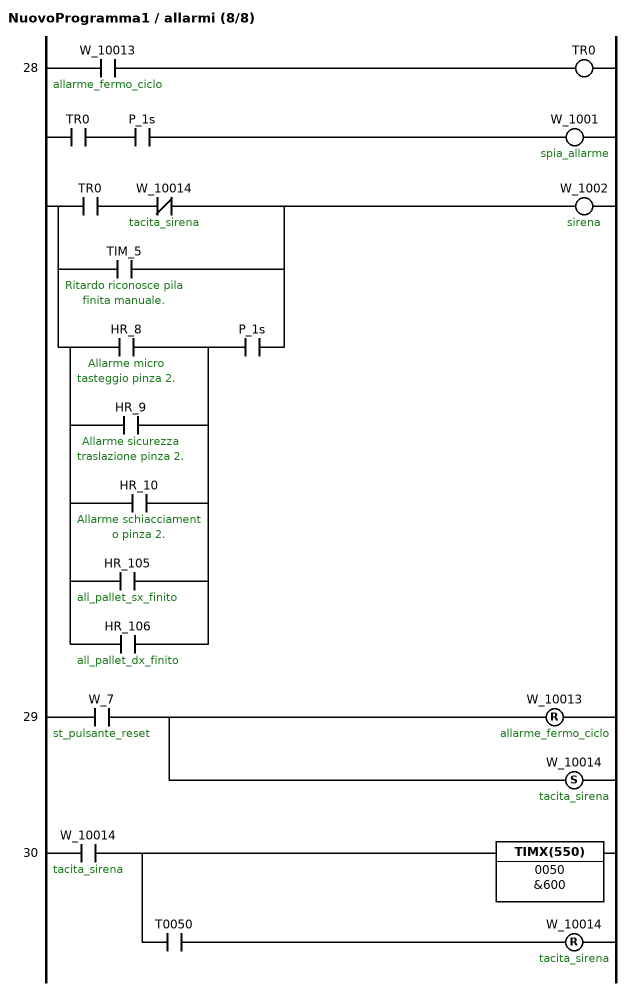
; rung 28
LD W_10013  ; allarme_fermo_ciclo
OUT TR0
AND P_1s
OUT W_1001  ; spia_allarme
LD TR0
ANDNOT W_10014  ; tacita_sirena
LD TIM_5  ; Ritardo riconosce pila finita manuale.
LD HR_8  ; Allarme micro tasteggio pinza 2.
OR HR_9  ; Allarme sicurezza traslazione pinza 2.
OR HR_10  ; Allarme schiacciamento pinza 2.
OR HR_105  ; all_pallet_sx_finito
OR HR_106  ; all_pallet_dx_finito
AND P_1s
ORLD
ORLD
OUT W_1002  ; sirena
; rung 29
LD W_7  ; st_pulsante_reset
RSET W_10013  ; allarme_fermo_ciclo
SET W_10014  ; tacita_sirena
; rung 30
LD W_10014  ; tacita_sirena
TIMX(550) 0050 &600
AND T0050
RSET W_10014  ; tacita_sirena

### Section velocità

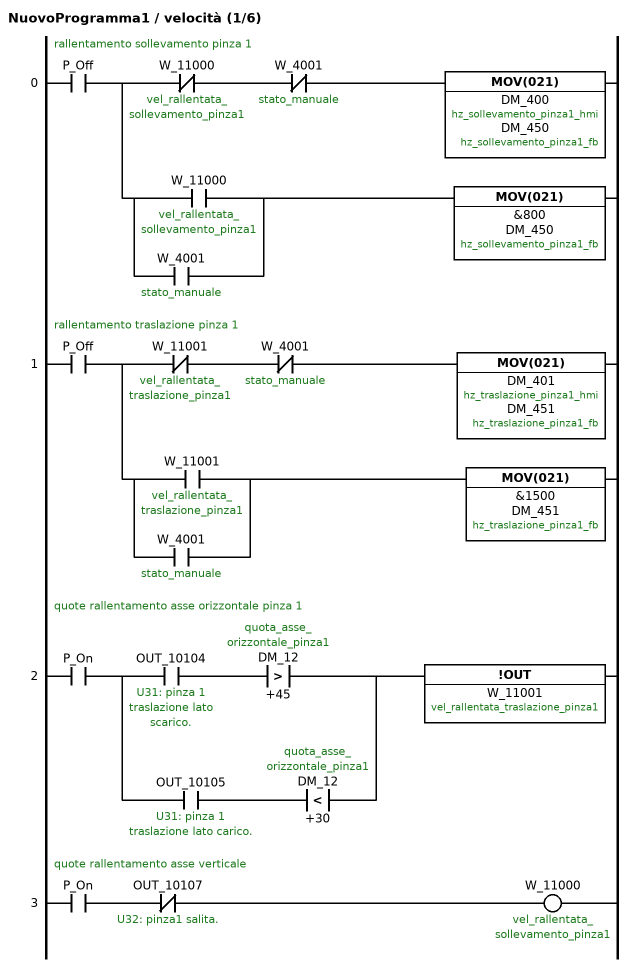
; rung 0: rallentamento sollevamento pinza 1
LD P_Off
OUT TR0
ANDNOT W_11000  ; vel_rallentata_sollevamento_pinza1
ANDNOT W_4001  ; stato_manuale
MOV(021) DM_400 DM_450  ; hz_sollevamento_pinza1_hmi, hz_sollevamento_pinza1_fb
LD TR0
LD W_11000  ; vel_rallentata_sollevamento_pinza1
OR W_4001  ; stato_manuale
ANDLD
MOV(021) &800 DM_450  ; hz_sollevamento_pinza1_fb
; rung 1: rallentamento traslazione pinza 1
LD P_Off
OUT TR0
!ANDNOT W_11001  ; vel_rallentata_traslazione_pinza1
ANDNOT W_4001  ; stato_manuale
MOV(021) DM_401 DM_451  ; hz_traslazione_pinza1_hmi, hz_traslazione_pinza1_fb
LD TR0
!LD W_11001  ; vel_rallentata_traslazione_pinza1
OR W_4001  ; stato_manuale
ANDLD
MOV(021) &1500 DM_451  ; hz_traslazione_pinza1_fb
; rung 2: quote rallentamento asse orizzontale pinza 1
LD P_On
!LD OUT_10104  ; U31: pinza 1 traslazione lato scarico.
AND>S(322) DM_12 +45  ; quota_asse_orizzontale_pinza1
!LD OUT_10105  ; U31: pinza 1 traslazione lato carico.
AND<S(312) DM_12 +30  ; quota_asse_orizzontale_pinza1
ORLD
ANDLD
!OUT W_11001  ; vel_rallentata_traslazione_pinza1
; rung 3: quote rallentamento asse verticale
LD P_On
ANDNOT OUT_10107  ; U32: pinza1 salita.
OUT W_11000  ; vel_rallentata_sollevamento_pinza1

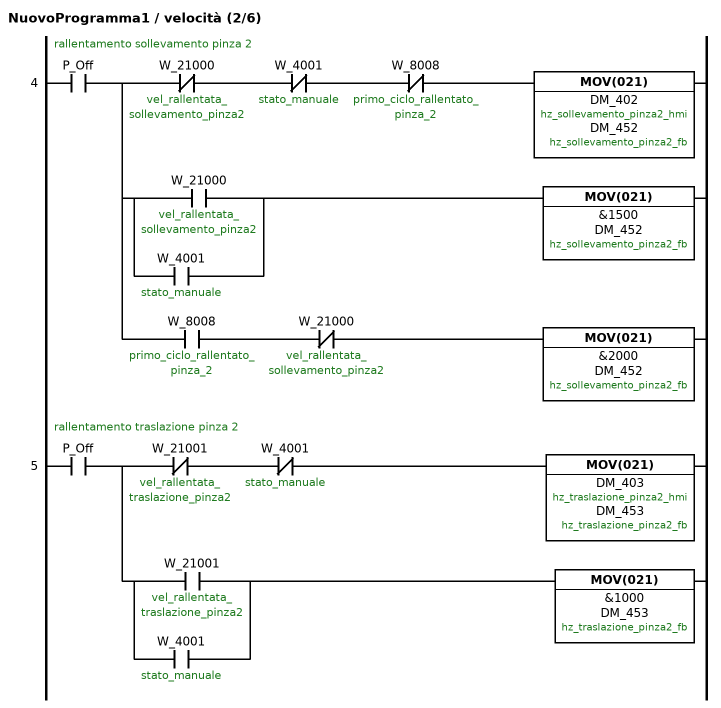
; rung 4: rallentamento sollevamento pinza 2
LD P_Off
OUT TR0
ANDNOT W_21000  ; vel_rallentata_sollevamento_pinza2
ANDNOT W_4001  ; stato_manuale
ANDNOT W_8008  ; primo_ciclo_rallentato_pinza_2
MOV(021) DM_402 DM_452  ; hz_sollevamento_pinza2_hmi, hz_sollevamento_pinza2_fb
LD TR0
LD W_21000  ; vel_rallentata_sollevamento_pinza2
OR W_4001  ; stato_manuale
ANDLD
MOV(021) &1500 DM_452  ; hz_sollevamento_pinza2_fb
LD TR0
AND W_8008  ; primo_ciclo_rallentato_pinza_2
ANDNOT W_21000  ; vel_rallentata_sollevamento_pinza2
MOV(021) &2000 DM_452  ; hz_sollevamento_pinza2_fb
; rung 5: rallentamento traslazione pinza 2
LD P_Off
OUT TR0
ANDNOT W_21001  ; vel_rallentata_traslazione_pinza2
ANDNOT W_4001  ; stato_manuale
MOV(021) DM_403 DM_453  ; hz_traslazione_pinza2_hmi, hz_traslazione_pinza2_fb
LD TR0
LD W_21001  ; vel_rallentata_traslazione_pinza2
OR W_4001  ; stato_manuale
ANDLD
MOV(021) &1000 DM_453  ; hz_traslazione_pinza2_fb

